FUNCTION_BLOCK fb_getCav
VAR_INPUT
	in_flg_run: BOOL;
END_VAR
VAR_OUTPUT
	out_flg_run: BOOL;
	out_flg_Done: BOOL;
	out_flg_error: BOOL;
	out_var_cav: INT;
END_VAR
VAR
	var_iCav : INT;
	fbi_r_trig: R_TRIG;
	var_process: INT;
END_VAR

out_flg_run := in_flg_run;
fbi_r_trig(CLK:=in_flg_run , Q=> );
IF fbi_r_trig.Q THEN
	var_process := 1;
END_IF
CASE var_process OF
	0:
			
	1:
		var_iCav.0 := gvl_io.flg_bitNumber0;
		var_iCav.1 := gvl_io.flg_bitNumber1;
		var_iCav.2 := gvl_io.flg_bitNumber2;
		var_iCav.3 := gvl_io.flg_bitNumber3;
		out_var_cav := var_iCav;
		var_process := 2;
	2:
		IF out_var_cav > gvl_param.var_productInfo[gvl_param.var_currentProductID].cavQty  OR out_var_cav = 0 THEN
			out_flg_error := TRUE;
			var_process := 4;
		ELSE
			var_process := 3;
		END_IF
	3:
		out_flg_Done := TRUE;
		var_process := 4;
	4:
		out_flg_error := FALSE;
		out_flg_Done := FALSE;
		var_process := 0;
END_CASE

END_FUNCTION_BLOCK

(* stored: Version 1.1.0.1, ProductVersion 3.1.4024.11
   POU fb_getCav: Id {92ace77b-bb30-4338-b21e-26db9bae8a7a}, SpecialFunc None *)
